TYPE Points :
STRUCT
	x:LREAL;
	y:LREAL;
	
END_STRUCT
END_TYPE

(* stored: Version 1.1.0.1, ProductVersion 3.1.4024.13
   DUT Points: Id {04a85ac3-3aa1-4172-a364-7898c67b7dfd} *)
